(* PLC project axle, Dassault Systèmes ControlBuild 2024x *)
(* stored: creationDateTime 2023-10-03T11:13:21-01:00 *)

(* This module simulates the behaviour of a limited axle to which a translation speed is imparted. *)
FUNCTION_BLOCK equipment_library.axle
  VAR_INPUT
    speed : REAL := 0.0;
  END_VAR
  VAR_OUTPUT
    positionTranslat : REAL := 0.0;
    percentTranslat : REAL := 0.0;
    incTranslat : REAL := 0.0;
  END_VAR
  VAR
    firstCycle : BOOL := false;
    nbCyclePerSec : REAL := 0.0;
  END_VAR
  VAR CONSTANT
    initTranslat : REAL := 0.0;
    maxTranslat : REAL := 10000.0;
    minTranslat : REAL := 0.0;
  END_VAR
  VAR
    d_locking : BOOL := false;
    v_d_locking : BOOL := false;
  END_VAR


ACTION C_source_code:
/* ----------------------------------------------------------------	*/
/* Type : Model of Operative Behaviour					*/
/* Category :  Actuators							*/
/* Author : Dassault Systemes						*/
/* Update date : June 2018							*/
/* ----------------------------------------------------------------	*/
/* This module simulates the behaviour of a limited axle to which a	*/
/* to which a translation speed is imparted.				*/
/* ----------------------------------------------------------------	*/

/* ----------------------------------------------------------------	*/
/* Initialise the position of the axle for the first step of 		*/
/* simulation.								*/
/* ----------------------------------------------------------------	*/
if ( ! firstCycle) {
	if (initTranslat > maxTranslat) positionTranslat = maxTranslat;
	else if (initTranslat < minTranslat) positionTranslat = minTranslat;
		else positionTranslat = initTranslat;
	firstCycle = 1;
}

/* -----------------------------------------------------------------	*/
/* Translation of the axle							*/
/* -----------------------------------------------------------------	*/

/* compute the increment of translation according to the simulation clock	*/
incTranslat = 0.0;
if (! d_locking) {
	nbCyclePerSec = CLOCK_PERIOD/1000000;
	incTranslat = speed * nbCyclePerSec;
}
positionTranslat = positionTranslat + incTranslat;

/* -----------------------------------------------------------------	*/
/* Limitation of the translation of the axle 				*/
/* -----------------------------------------------------------------	*/
if (positionTranslat > maxTranslat) {
	incTranslat -= positionTranslat - maxTranslat;
	positionTranslat = maxTranslat;
}
if (positionTranslat < minTranslat) {
	incTranslat -= positionTranslat - minTranslat;
	positionTranslat = minTranslat;
}

/* ----------------------------------------------------------------- */
/* Compute the percent between the position and the limit		*/
/* ----------------------------------------------------------------- */

percentTranslat = (100/(maxTranslat - minTranslat)) * (positionTranslat - minTranslat)  ;
		
END_ACTION
END_FUNCTION_BLOCK
